{attribute 'GeneratedUsingTerminal: EL6001-0000-0020'}
{attribute addProperty BoxType "EL6001-0000-0020"}
{attribute addProperty Id "COM_InputsAT %I*COM_Inputs_3801C95E30COM_OutputsAT %Q*COM_Outputs_DEF408EC27WcStateAT %I*WcState_9091E0EB2InfoDataAT %I*InfoData_94A18F5E2"}
{attribute addProperty CRC "74562978"}
{attribute addProperty Size "61"}
TYPE EL6001_0471BDA2 EXTENDS EtcSlaveTerminalBase_947E5A46 :
STRUCT
	{attribute addProperty Name "COM_Inputs"}
	COM_Inputs : COM_Inputs_3801C95E;
	{attribute addProperty Name "COM_Outputs"}
	COM_Outputs : COM_Outputs_DEF408EC;
	{attribute addProperty Name "WcState"}
	WcState : WcState_9091E0EB;
	{attribute addProperty Name "InfoData"}
	InfoData : InfoData_94A18F5E;
END_STRUCT
END_TYPE

(* stored: Version 1.2.0.0, ProductVersion 3.1.4024.9
   DUT EL6001_0471BDA2: Id {d0ea15d4-96d0-42ee-8e3b-cd69761c92d1} *)
